FUNCTION proj1_TupleStruct_2: LREAL
VAR_INPUT
    tuple: TupleStruct_2;
END_VAR


        proj1_TupleStruct_2 := tuple.field1;

END_FUNCTION

(* stored: ProductVersion 3.1.0.18, Version 1.1.0.1 *)
